Xinje XCPPro project, PLC1: XC3-24 (software 3.3L)

PROGRAM Ladder

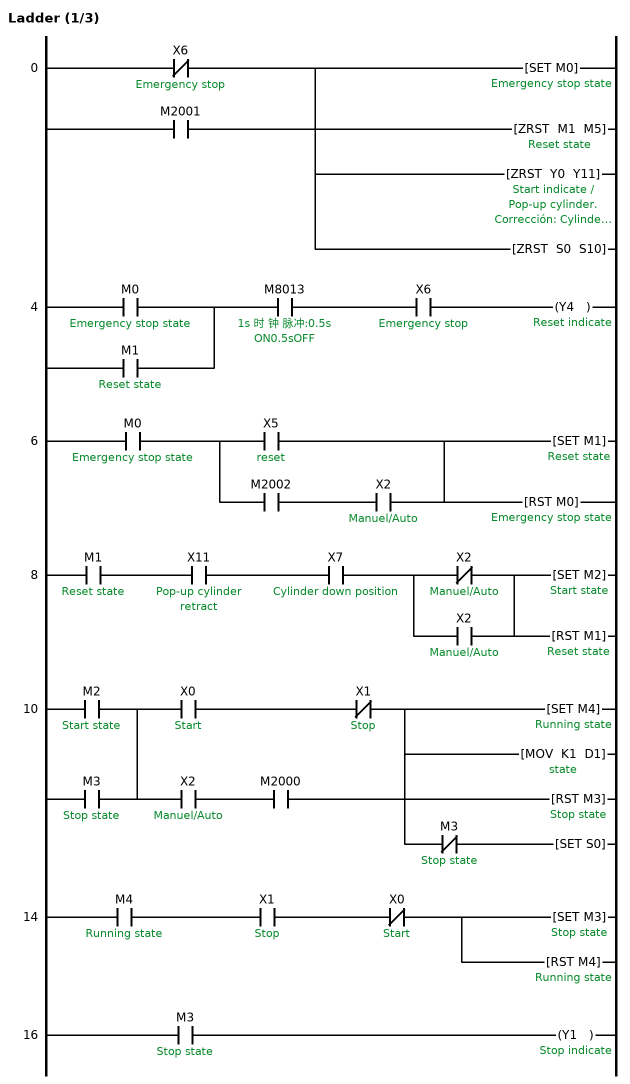
LDI    X6	; Emergency stop
OR     M2001
SET    M0	; Emergency stop state
ZRST   M1 M5	; Reset state
ZRST   Y0 Y11	; Start indicate / Pop-up cylinder. Corrección: Cylinder down.
ZRST   S0 S10
LD     M0	; Emergency stop state
OR     M1	; Reset state
AND    M8013	; 1s 时 钟 脉冲:0.5s ON0.5sOFF
AND    X6	; Emergency stop
OUT    Y4	; Reset indicate 
LD     M0	; Emergency stop state
LD     X5	; reset
LD     M2002
AND    X2	; Manuel/Auto
ORB
ANB
SET    M1	; Reset state
RST    M0	; Emergency stop state
LD     M1	; Reset state
AND    X11	; Pop-up cylinder retract 
AND    X7	; Cylinder down position 
LDI    X2	; Manuel/Auto
OR     X2	; Manuel/Auto
ANB
SET    M2	; Start state
RST    M1	; Reset state
LD     M2	; Start state
OR     M3	; Stop state
LD     X0	; Start
ANI    X1	; Stop
LD     X2	; Manuel/Auto
AND    M2000
ORB
ANB
SET    M4	; Running state
MOV    K1 D1	; state
RST    M3	; Stop state
ANI    M3	; Stop state
SET    S0
LD     M4	; Running state
AND    X1	; Stop
ANI    X0	; Start
SET    M3	; Stop state
RST    M4	; Running state
LD     M3	; Stop state
OUT    Y1	; Stop indicate

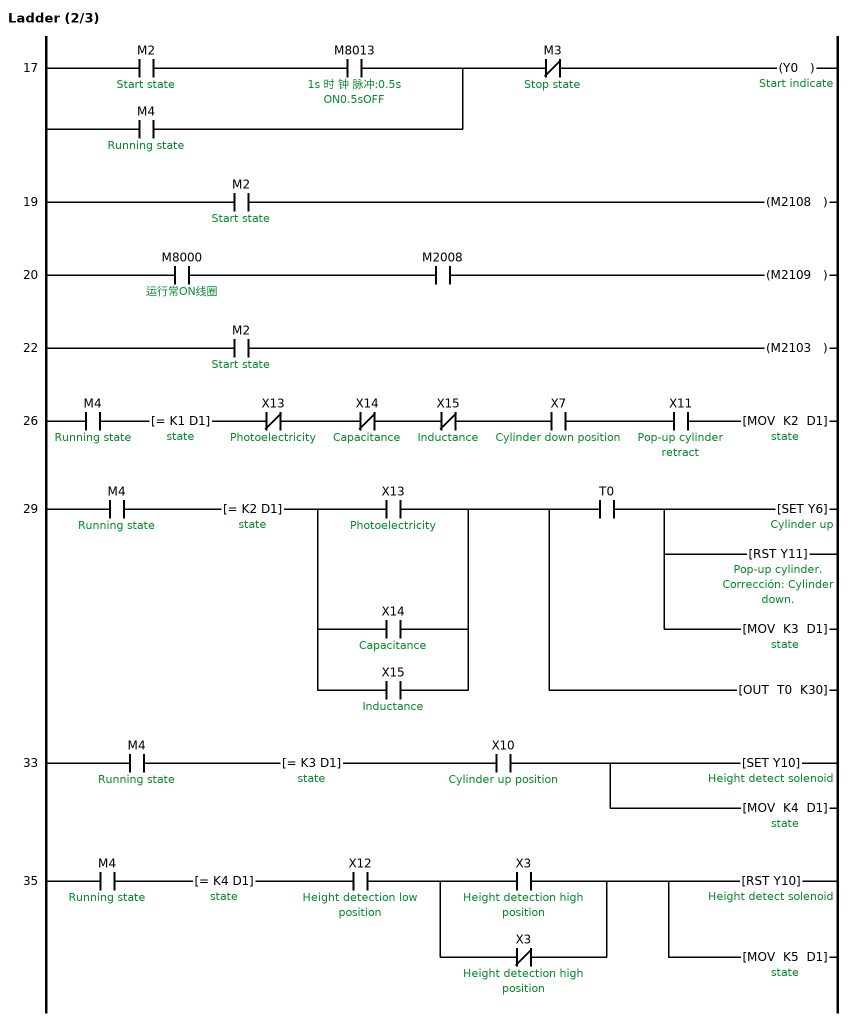
LD     M2	; Start state
AND    M8013	; 1s 时 钟 脉冲:0.5s ON0.5sOFF
OR     M4	; Running state
ANI    M3	; Stop state
OUT    Y0	; Start indicate
LD     M2	; Start state
OUT    M2108
LD     M8000	; 运行常ON线圈
AND    M2008
OUT    M2109
LD     M2	; Start state
OUT    M2103
LD     M4	; Running state
AND=   K1 D1	; state
ANI    X13	; Photoelectricity
ANI    X14	; Capacitance
ANI    X15	; Inductance
AND    X7	; Cylinder down position 
AND    X11	; Pop-up cylinder retract 
MOV    K2 D1	; state
LD     M4	; Running state
AND=   K2 D1	; state
LD     X13	; Photoelectricity
OR     X14	; Capacitance
OR     X15	; Inductance
ANB
MPS
AND    T0
SET    Y6	; Cylinder up 
RST    Y11	; Pop-up cylinder. Corrección: Cylinder down.
MOV    K3 D1	; state
MPP
OUT    T0 K30
LD     M4	; Running state
AND=   K3 D1	; state
AND    X10	; Cylinder up position
SET    Y10	; Height detect solenoid
MOV    K4 D1	; state
LD     M4	; Running state
AND=   K4 D1	; state
AND    X12	; Height detection low position
LD     X3	; Height detection high position 
ORI    X3	; Height detection high position 
ANB
RST    Y10	; Height detect solenoid
MOV    K5 D1	; state

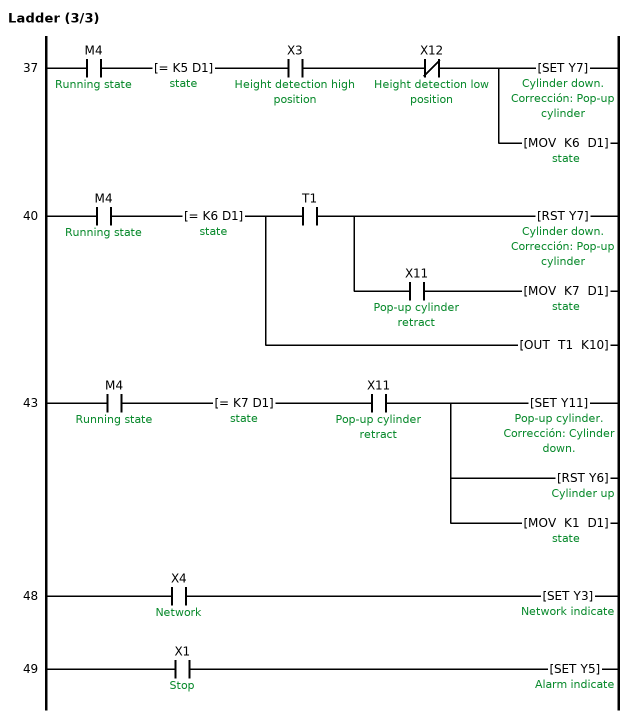
LD     M4	; Running state
AND=   K5 D1	; state
AND    X3	; Height detection high position 
ANI    X12	; Height detection low position
SET    Y7	; Cylinder down. Corrección: Pop-up cylinder
MOV    K6 D1	; state
LD     M4	; Running state
AND=   K6 D1	; state
MPS
AND    T1
RST    Y7	; Cylinder down. Corrección: Pop-up cylinder
AND    X11	; Pop-up cylinder retract 
MOV    K7 D1	; state
MPP
OUT    T1 K10
LD     M4	; Running state
AND=   K7 D1	; state
AND    X11	; Pop-up cylinder retract 
SET    Y11	; Pop-up cylinder. Corrección: Cylinder down.
RST    Y6	; Cylinder up 
MOV    K1 D1	; state
LD     X4	; Network
SET    Y3	; Network indicate
LD     X1	; Stop
SET    Y5	; Alarm indicate